# EPICS autosave request: dxp/trunk/dxpApp/Db/dxp_settings.req
# FILE... dxp_settings.req
# USAGE.. dxp2x.db or dxp4c.db fields autosave'd.
$(P)$(R).SCAN
$(P)$(R).PGAIN
$(P)$(R).SLOW_TRIG
$(P)$(R).PKTIM
$(P)$(R).GAPTIM
$(P)$(R).FAST_TRIG
$(P)$(R).TRIG_PKTIM
$(P)$(R).TRIG_GAPTIM
$(P)$(R).ADC_RULE
$(P)$(R).EMAX
$(P)$(R).TRACE_WAIT
